FUNCTION TorrToMbarWithAlias : mbar
VAR_INPUT
    pressure : Torr;
END_VAR

TorrToMbarWithAlias := pressure * 1.3332236842;

END_FUNCTION

(* stored: Version 1.1.0.1, ProductVersion 3.1.4024.4
   POU TorrToMbarWithAlias: Id {ddfc8f5b-03ad-43e0-85dd-c1361620af61}, SpecialFunc None *)
